// TIA Portal V19 export
TYPE "C402_STU_AFS_IF_SBO_TYPIC"
   STRUCT
      CMD_HND { ExternalAccessible := 'False'; ExternalVisible := 'False'; ExternalWritable := 'False'} : Bool;   // Commando Bedieningsmode Hand activeren
      CMD_OPEN { ExternalAccessible := 'False'; ExternalVisible := 'False'; ExternalWritable := 'False'} : Bool;   // Commando Openen afsluitboom (voor hulpdiensten)
      STS_VKL_OK { ExternalAccessible := 'False'; ExternalVisible := 'False'; ExternalWritable := 'False'} : Bool;   // 1 = Verkeerslichten op Rood
      EXT_STO { ExternalAccessible := 'False'; ExternalVisible := 'False'; ExternalWritable := 'False'} : Bool;   // Externe storing aanwezig
      EXT_NDS_NOK { ExternalAccessible := 'False'; ExternalVisible := 'False'; ExternalWritable := 'False'} : Bool;   // Noodstopkring niet in orde
   END_STRUCT;
END_TYPE
